// TwinCAT 3 PLC project File
// Title: ZigaLibs.File
// Company: Ziga Javornik
// Author: Ziga Javornik
// ProjectVersion: 0.2.2.0
// Description: Library containing logic for file handling and helper programs.
// ProgramVersion: 3.1.4026.26
// libraries:
//   Tc2_Standard, * (Beckhoff Automation GmbH)
//   Tc2_System, * (Beckhoff Automation GmbH)
//   Tc2_Utilities, * (Beckhoff Automation GmbH)
//   Tc3_Module, * (Beckhoff Automation GmbH)
//   TcError, * (Roald87)
//   TcUnit, * (www.tcunit.org)
//   ZigaLibs.Core, * (Ziga Javornik)
// project tree:
//   SOURCE/Constants/ Constants.TcPOU, FB_PathSeperators.TcPOU, FB_Wildcards.TcPOU
//   SOURCE/DUTs/ E_FileOpenMode.TcDUT, ST_FileInfo.TcDUT, T_FileAccessMode.TcDUT, T_FileHandle.TcDUT
//   SOURCE/Utilities/Directory/ E_DeleteFilesByDateState.TcDUT, E_GetFilesState.TcDUT, FB_DirectoryUtilities.TcPOU, I_Directory.TcIO
//   SOURCE/Utilities/File/ FB_FileUtilities.TcPOU, I_File.TcIO
//   SOURCE/Utilities/Path/ FB_PathGenerator.TcPOU, FB_PathUtilities.TcPOU, I_Path.TcIO, I_PathGenerator.TcIO, I_Wildcards.TcIO
//   SOURCE/FileHandler/ FB_FileHandler.TcPOU, I_FileHandler.TcIO, I_FileProperties.TcIO
//   SOURCE/Utilities/ Utilities.TcPOU
//   / TestsTask.TcTTO
//   TESTS/ PRG_TESTS.TcPOU
//   TESTS/Test suites/ FB_DirectoryUtilities_Tests.TcPOU, FB_FileHandler_Tests.TcPOU, FB_FileUtilities_Tests.TcPOU, FB_Utilities_Tests.TcPOU, FB_PathGenerator_Tests.TcPOU, FB_PathUtilities_Tests.TcPOU
// (motion and I/O tree: see PLC project logging)
// real-time tasks:
//   TASK TestsTask: cycle T#10ms, priority 20, ADS port 350
//   TASK PlcTask: cycle T#10ms, priority 21, ADS port 351

CONFIGURATION File
    RESOURCE PLC ON TwinCAT3
        TASK TestsTask(INTERVAL := T#10ms, PRIORITY := 20);
        PROGRAM PRG_TESTS WITH TestsTask : PRG_TESTS;
    END_RESOURCE
END_CONFIGURATION

// ---- SOURCE/DUTs/E_FileOpenMode.TcDUT
// A combination of file open modes, based on available options.
// Source: https://infosys.beckhoff.com/english.php?content=../content/1033/tcplclib_tc2_system/30977547.html&id=
{attribute 'strict'}
{attribute 'to_string'}
TYPE E_FileOpenMode :
(
	(* r: Opens a file for reading. An error is returned if the file cannot be found or does not exist.*)
	TEXT_READ_MUST_EXIST := Tc2_System.FOPEN_MODEREAD OR Tc2_System.FOPEN_MODETEXT,
	
	(* 	w: Opens an empty file for writing. If the file already exists, it is overwritten.*)
	TEXT_WRITE_OVERWRITE_EXISTING := Tc2_System.FOPEN_MODEWRITE OR Tc2_System.FOPEN_MODETEXT,
	
	(* a: Opens a file for writing at the end of the file (append). If the file does not exist, a new file is created.*)
	TEXT_APPEND := Tc2_System.FOPEN_MODEAPPEND OR Tc2_System.FOPEN_MODETEXT,
	
	(* r+: Opens a file for reading and writing. The file must exist.*)
	TEXT_READ_WRITE_MUST_EXIST := Tc2_System.FOPEN_MODEREAD OR Tc2_System.FOPEN_MODEPLUS OR Tc2_System.FOPEN_MODETEXT,
	
	(* w+: Opens an empty file for reading and writing. If the file already exists, it is overwritten.*)
	TEXT_READ_WRITE_OVERWRITE_EXISTING := Tc2_System.FOPEN_MODEWRITE OR Tc2_System.FOPEN_MODEPLUS OR Tc2_System.FOPEN_MODETEXT,
	
	(* a+: opens a file for reading and writing at the end of the file (append). 
	If the file does not exist, a new file is created. For this, the memory path must be known, otherwise error 1804 appears. 
	All write operations are always performed at end of a file, if the file was opened in the modes a or a+.
	The file pointer can be moved with FB_FileSeek, although for writing it is moved to the end of the file by default, i.e. existing data cannot be overwritten.*)
	TEXT_READ_WRITE_APPEND	:= Tc2_System.FOPEN_MODEAPPEND OR Tc2_System.FOPEN_MODEPLUS OR Tc2_System.FOPEN_MODETEXT,
	
	(* r: Opens a file for reading. An error is returned if the file cannot be found or does not exist.*)
	BINARY_READ_MUST_EXIST	:= Tc2_System.FOPEN_MODEREAD OR Tc2_System.FOPEN_MODEBINARY,
	
	(* 	w: Opens an empty file for writing. If the file already exists, it is overwritten.*)
	BINARY_WRITE_OVERWRITE_EXISTING := Tc2_System.FOPEN_MODEWRITE OR Tc2_System.FOPEN_MODEBINARY,
	
	(* a: Opens a file for writing at the end of the file (append). If the file does not exist, a new file is created.*)
	BINARY_APPEND := Tc2_System.FOPEN_MODEAPPEND OR Tc2_System.FOPEN_MODEBINARY,
	
	(* r+: Opens a file for reading and writing. The file must exist.*)
	BINARY_READ_WRITE_MUST_EXIST := Tc2_System.FOPEN_MODEREAD OR Tc2_System.FOPEN_MODEPLUS OR Tc2_System.FOPEN_MODEBINARY,
	
	(* w+: Opens an empty file for reading and writing. If the file already exists, it is overwritten.*)
	BINARY_READ_WRITE_OVERWRITE_EXISTING := Tc2_System.FOPEN_MODEWRITE OR Tc2_System.FOPEN_MODEPLUS OR Tc2_System.FOPEN_MODEBINARY,
	
	(* a+: opens a file for reading and writing at the end of the file (append). 
	If the file does not exist, a new file is created. For this, the memory path must be known, otherwise error 1804 appears. 
	All write operations are always performed at end of a file, if the file was opened in the modes a or a+.
	The file pointer can be moved with FB_FileSeek, although for writing it is moved to the end of the file by default, i.e. existing data cannot be overwritten.*)
	BINARY_READ_WRITE_APPEND := Tc2_System.FOPEN_MODEAPPEND OR Tc2_System.FOPEN_MODEPLUS OR Tc2_System.FOPEN_MODEBINARY
)DWORD;
END_TYPE

// ---- SOURCE/DUTs/ST_FileInfo.TcDUT
// Structure with all the information for working with file handling..
TYPE ST_FileInfo :
STRUCT
	Handle 		: T_FileHandle;				// File handle
	NetId		: Tc2_System.T_AmsNetID;	// NetId where the file is located
	Name		: Tc2_System.T_MaxString;	// Name of the file
	Path		: Tc2_System.T_MaxString;	// Locaiton of the file
	IsOpened	: BOOL;
END_STRUCT
END_TYPE

// ---- SOURCE/DUTs/T_FileAccessMode.TcDUT
TYPE T_FileAccessMode : DWORD; END_TYPE

// ---- SOURCE/DUTs/T_FileHandle.TcDUT
TYPE T_FileHandle : UINT; END_TYPE

// ---- SOURCE/Utilities/Directory/E_DeleteFilesByDateState.TcDUT
{attribute 'qualified_only'}
{attribute 'strict'}
TYPE E_DeleteFilesByDateState :
(
	START,
	GET_FILE,
	WAIT_FOR_DELETE
);
END_TYPE

// ---- SOURCE/Utilities/Directory/E_GetFilesState.TcDUT
{attribute 'qualified_only'}
{attribute 'strict'}
TYPE INTERNAL E_GetFilesState :
(
	READY,
	START,
	AWAIT_RESULT,
	ALL_FILES_FOUND,
	ERROR
);
END_TYPE

// ---- SOURCE/Utilities/Directory/I_Directory.TcIO
INTERFACE I_Directory

// Deletes files in the directory that were created before the provided date.
METHOD DeleteFilesCreatedBefore : BOOL
VAR_INPUT
	path				: Tc2_System.T_MaxString;	// Path to where the deletion should be performed
	fileNameContains	: Tc2_System.T_MaxString;	// Some characters that the file name should containt
	netId				: Tc2_System.T_AmsNetID;	// NetId where the search should occurr
	thresholdDate		: DT;	// If created before this date, the file will be deleted.
END_VAR

VAR_OUTPUT
	error			: BOOL;
	errorInfo		: ZigaLibs_Core.ST_AdsError;	
	deletedFiles	: ARRAY[0..100] OF Tc2_System.T_MaxString;	// A list of deleted items, as T_MaxString (file names).
END_VAR
END_METHOD

// Looks if the provided directory exists on the disk.
// Returns TRUE when done
// Result can be found in the output directoryExists.
METHOD Exists : BOOL
VAR_INPUT
	directory	: Tc2_System.T_MaxString;	// Path to the directory that will be searched.
	netId		: Tc2_System.T_AmsNetID;	// NetId where to search.
END_VAR

VAR_OUTPUT
	directoryExists		: BOOL;	// TRUE if it exists, else FALSE. Only valid after method returns TRUE.
END_VAR
END_METHOD

(* Looks in the directory `path` and iterates the content. 
 When method returns TRUE, the collection of items is found in the result I_Collection.*)
METHOD ListAll : BOOL
VAR_INPUT
	path	: Tc2_System.T_MaxString;	// Path to the directory that will be searched.
	netId	: Tc2_System.T_AmsNetID;	// NetId where to search.
END_VAR

VAR_IN_OUT
	items	: ARRAY[*] OF Tc2_Utilities.ST_FindFileEntry;	// Collection of found files in the provided location	
END_VAR

VAR_OUTPUT
	error		: BOOL;	// Will be true if an error occurs while executing the file query
	errorInfo	: ZigaLibs_Core.ST_AdsError;	// Error information will be provided here
END_VAR
END_METHOD

(* Looks in the directory `path` and iterates the content. 
 When method returns TRUE, the collection of files is found in the result I_Collection.*)
METHOD ListFiles : BOOL
VAR_INPUT
	path	: Tc2_System.T_MaxString;	// Path to the directory that will be searched.
	netId	: Tc2_System.T_AmsNetID;	// NetId where to search.
END_VAR

VAR_IN_OUT
	files	: ARRAY[*] OF Tc2_System.T_MaxString;	// Collection of found files in the provided location.
END_VAR

VAR_OUTPUT
	error		: BOOL;	// Will be true if an error occurs while executing the file query
	errorInfo	: ZigaLibs_Core.ST_AdsError;	// Error information will be provided here
END_VAR
END_METHOD

END_INTERFACE

// ---- SOURCE/Utilities/File/I_File.TcIO
INTERFACE I_File

METHOD Create : BOOL
VAR_INPUT
	path		: Tc2_System.T_MaxString;	// Path to where the file will be created
	name		: Tc2_System.T_MaxString;	// Name of the file to create.
	netId		: Tc2_System.T_AmsNetID;	// NetId of the device where the file will be created
	overwrite	: BOOL;						// If set to TRUE, if the file with the provided name already exists, it will be overwritten
END_VAR
VAR_OUTPUT
	error			: BOOL;
	errorInfo	: ZigaLibs_Core.ST_AdsError;
END_VAR
END_METHOD

// Deletes the file. Returns TRUE when done.
METHOD Delete : BOOL
VAR_INPUT
	path	: Tc2_System.T_MaxString;	// Location of the file
	name	: Tc2_System.T_MaxString;	// File to be deleted
	netId	: Tc2_System.T_AmsNetID;
END_VAR
VAR_OUTPUT
	error			: BOOL;
	errorInfo	: ZigaLibs_Core.ST_AdsError;
END_VAR
END_METHOD

// Checks the content at `path` and looks for the file with `name`. Returns TRUE when done. 
// If file exissts, the result ˛`result` will be TRUE, else it will be fALSE.
METHOD Exists : BOOL
VAR_INPUT
	path	: Tc2_System.T_MaxString;	// Path to the file location
	name	: Tc2_System.T_MaxString;	// Name of the file
	netId	: Tc2_System.T_AmsNetID;	// NetId where the file is located
END_VAR

VAR_OUTPUT
	result		: BOOL; // Result, if the file exists or not - check when method returns TRUE
	error		: BOOL;	// Will be true if an error occurs while executing the file query
	errorInfo	: ZigaLibs_Core.ST_AdsError; // Error information will be provided here
END_VAR
END_METHOD

END_INTERFACE

// ---- SOURCE/Utilities/Path/I_Path.TcIO
INTERFACE I_Path

(* Checks if path exists, return TRUE when done and the result is returned in `result` output var.*)
METHOD Exists : BOOL
VAR_INPUT
	path	: Tc2_System.T_MaxString;
	netId	: Tc2_System.T_AmsNetID;
END_VAR

VAR_OUTPUT
	result		: BOOL; // Result, if the file exists or not - check when method returns TRUE
	error		: BOOL;	// Will be true if an error occurs while executing the file query
	errorInfo	: ZigaLibs_Core.ST_AdsError; // Error information will be provided here
END_VAR
END_METHOD

(* Generates the file path based on the location, file name and extension*)
METHOD Generate : I_PathGenerator
END_METHOD

END_INTERFACE

// ---- SOURCE/Utilities/Path/I_PathGenerator.TcIO
INTERFACE I_PathGenerator

METHOD AddWildcard : I_Wildcards
VAR_INPUT
END_VAR
END_METHOD

METHOD Create : T_MaxString
VAR_INPUT
END_VAR
END_METHOD

// Concatines the path with previously added paths. 
// If the provided path does not starts with the system-based path seperator, it is added

// Example:
// Join('C:/Program Files/').Join('Utilities/SystemUtilities') 
// will result in 'C:/Program Files/Utilities/SystemUtilities'
METHOD Join : I_PathGenerator
VAR_INPUT
	path	: STRING;
END_VAR
END_METHOD

END_INTERFACE

// ---- SOURCE/Utilities/Path/I_Wildcards.TcIO
INTERFACE I_Wildcards

METHOD Asterisk : I_PathGenerator
VAR_INPUT
	left	: Tc2_System.T_MaxString;
	right	: Tc2_System.T_MaxString;
END_VAR
END_METHOD

METHOD Questionmark : I_PathGenerator
VAR_INPUT
END_VAR
END_METHOD

END_INTERFACE

// ---- SOURCE/FileHandler/I_FileHandler.TcIO
INTERFACE I_FileHandler EXTENDS I_FileProperties

// Closes the file and returns TRUE when done.
METHOD Close : BOOL
END_METHOD

// Creates the file
METHOD Create : BOOL
VAR_INPUT
	path	: Tc2_System.T_MaxString;	// Path to the file location
	name	: Tc2_System.T_MaxString;	// Name of the file
	netId	: Tc2_System.T_AmsNetID;	// NetId where the file is located
END_VAR
END_METHOD

// Flushes the current file stream data to the file. 
// Basically file is closed and re-opened, which in turn writes the content of the stream to the file.
// If the file was opened to overwrite existing content, flushing will clear the data in the file!
// While flushing is being executed, the .File property DOES NOT CHANGE 
// For example, the File.IsOpened will remain TRUE even at the point where it is actually not. It will then be re-opened. 
// If an error occurs however, properties will be set to correct state.

METHOD Flush : BOOL
END_METHOD

// Opens the file in the path provided. If a file is already opened nothing happens.
// Returns: TRUE when done.
METHOD Open : BOOL
VAR_INPUT
	path	: Tc2_System.T_MaxString;	// Path to the file location
	name	: Tc2_System.T_MaxString;	// Name of the file
	mode	: E_FileOpenMode;			// Mode in which the file will be opened
	netId	: Tc2_System.T_AmsNetID;	// NetId where the file is located
END_VAR
END_METHOD

// Opens the last file with the provided open parameters. 
// If file can't be opened or no file has been opened so far, an error is gnerated.
METHOD OpenLast : BOOL
END_METHOD

// Reads the file and writes the content to the result variable.
// Resturns TRUE when done.
METHOD Read : BOOL
VAR_INPUT
	result	: ANY;
END_VAR
END_METHOD

// Reset any existing error.
METHOD Reset
END_METHOD

(* Returns TRUE if there is no content in the file stream.*)
{attribute'monitoring':='call'}
PROPERTY StreamEmpty : BOOL
GET
END_GET
END_PROPERTY

// Writes binary content to the file.
// Returns TRUE when done.
METHOD WriteBinary : BOOL
VAR_INPUT
	data		: ANY;	// Bincary content to be written
END_VAR
END_METHOD

// Writes a single line to the file
// Returns TRUE when done.
METHOD WriteLine : BOOL
VAR_INPUT
	line	: Tc2_System.T_MaxString;	// Text to be written
END_VAR
END_METHOD

END_INTERFACE

// ---- SOURCE/FileHandler/I_FileProperties.TcIO
// Provies interface to properties required for file access
INTERFACE I_FileProperties

{attribute 'monitoring':='call'}
// Gets or set file properties.
PROPERTY File : REFERENCE TO ST_FileInfo
GET
END_GET
END_PROPERTY

END_INTERFACE

// ---- TESTS/PRG_TESTS.TcPOU
PROGRAM INTERNAL PRG_TESTS

(* Instantiate test suites here. Naming convention for tests should be a suffix with _Tests.
Good practice for creating test methods is to end them with _test as well. *)
VAR
	PathGeneratorTests		: FB_PathGenerator_Tests;
	UtilitiesTests			: FB_Utilities_Tests;
	FileHandlerTests		: FB_FileHandler_Tests;
	PathUtilitiesTests		: FB_PathUtilities_Tests;
	FileUtilitiesTests		: FB_FileUtilities_Tests;
	DirectoryUtilitiesTests	: FB_DirectoryUtilities_Tests;
END_VAR

VAR CONSTANT
	FILE_HANDLER_TESTS_PATH			: Tc2_System.T_MaxString := '/home/Administrator/ZigaLibsTestFolder/FileHandlerTests/';
	FILE_HANDLER_TESTS_DIRECTORY	: Tc2_System.T_MaxString := '/home/Administrator/ZigaLibsTestFolder/FileHandlerTests';
	NET_ID							: Tc2_System.T_AmsNetID := '';
	DATE_TIME_MAX_VALUE				: DT  := DATE_AND_TIME#2106-02-07-06:28:15;
END_VAR

// Run tests in parallel
//TcUnit.RUN();

// Run tests in sequence, one after the other.
TcUnit.RUN_IN_SEQUENCE();

END_PROGRAM

// ---- TESTS/Test suites/FB_PathGenerator_Tests.TcPOU
FUNCTION_BLOCK INTERNAL FB_PathGenerator_Tests EXTENDS FB_TestSuite
VAR_INPUT
END_VAR
VAR_OUTPUT
END_VAR
VAR
	_pathGenerator	: FB_PathGenerator;
END_VAR

Test01_VariousPathOptions();

METHOD Test01_VariousPathOptions

// These test values were taken from microsoft Path.Join documentation at 
// https://learn.microsoft.com/en-us/dotnet/api/system.io.path.join?view=net-9.0
VAR
	path1 : STRING := 'C:/Program Files/';
	path2 : STRING := 'Utilities/SystemUtilities';
	expectedResult_path1_2	: STRING := 'C:/Program Files/Utilities/SystemUtilities';
	
	
	path3 : STRING := 'C:/';
	path4 : STRING := '/Program Files';
	expectedResult_path3_4	: STRING := 'C://Program Files';
	
	path5 : STRING := 'C:/Users/Public/Documents/';
	path6 : STRING := 'C:/Users/User1/Documents/Financial/';
	expectedResult_path5_6	: STRING := 'C:/Users/Public/Documents/C:/Users/User1/Documents/Financial/';	
END_VAR
TcUnit.TEST('Test01_VariousPathOptions');

AssertEquals_STRING(
	Expected := expectedResult_path1_2, 
	Actual := _pathGenerator.Join(path1).Join(path2).Create(),
	'Joining paths 1 and 2 failed.');
	
AssertEquals_STRING(
	Expected := expectedResult_path3_4, 
	Actual := _pathGenerator.Join(path3).Join(path4).Create(),
	'Joining paths 2 and 3 failed.');
	
AssertEquals_STRING(
	Expected := expectedResult_path5_6, 
	Actual := _pathGenerator.Join(path5).Join(path6).Create(),
	'Joining paths 4 and 5 failed.');
		
TcUnit.TEST_FINISHED();
END_METHOD

END_FUNCTION_BLOCK

// ---- SOURCE/Utilities/Path/FB_PathGenerator.TcPOU
FUNCTION_BLOCK FB_PathGenerator IMPLEMENTS I_PathGenerator, I_Wildcards
VAR_INPUT
END_VAR
VAR_OUTPUT
END_VAR
VAR
	_path			: Tc2_System.T_MaxString;
END_VAR

// Provides ability to add allowed wildcards to the generating path.
METHOD AddWildcard : I_Wildcards
AddWildcard := THIS^;
END_METHOD

// Adds the asterisk (*) wildcard between the left and right strings provided
// Example Asterix('abc','def') => '<path so far>abc*def'
METHOD Asterisk : I_PathGenerator
VAR_INPUT
	left	: Tc2_System.T_MaxString;
	right	: Tc2_System.T_MaxString;
END_VAR
ZigaLibs_Core.StringHelper.Join(left, Constants.Wildcards.Asterisk);
ZigaLibs_Core.StringHelper.Join(left, right);
ZigaLibs_Core.StringHelper.Join(_path, left);
Asterisk := THIS^;
END_METHOD

METHOD Create : Tc2_System.T_MaxString
Create := _path;
_path := '';
END_METHOD

// Concatines the path with previously added paths. 
// If the provided path does not starts with the system-based path seperator, it is added

// Example:
// Join('C:/Program Files/').Join('Utilities/SystemUtilities') 
// will result in 'C:/Program Files/Utilities/SystemUtilities'
METHOD Join : I_PathGenerator
VAR_INPUT
	path	: STRING;
END_VAR
Join := THIS^;

// If this is the root, skip adding seperator to start.
IF Tc2_Standard.FIND(path, ':') <> 0 THEN
	ZigaLibs_Core.StringHelper.Join(_path, path);
	RETURN;
END_IF

// Add path seperator, if not starting with it.
IF NOT ZigaLibs_Core.StringHelper.StartsWith(path, Constants.PathSeperators.Windows) AND
   NOT ZigaLibs_Core.StringHelper.EndsWith(_path, Constants.PathSeperators.Windows) AND
   NOT ZigaLibs_Core.StringHelper.StartsWith(path, Constants.PathSeperators.Unix) AND
   NOT ZigaLibs_Core.StringHelper.EndsWith(_path, Constants.PathSeperators.Unix)
THEN
	path := Tc2_Standard.CONCAT(Constants.PathSeperators.Independent, path);
END_IF
ZigaLibs_Core.StringHelper.Join(_path, path);
END_METHOD

// Adds the question mark (?) wildcard to the end of the currently generated path.
METHOD Questionmark : I_PathGenerator
ZigaLibs_Core.StringHelper.Join(_path, Constants.Wildcards.QuestionMark);
Questionmark := THIS^;
END_METHOD

END_FUNCTION_BLOCK

// ---- SOURCE/Constants/Constants.TcPOU
// Contains string constants for working with files
{attribute 'no_explicit_call' := 'Body contains no logic, calling methods only allowed.'}
{attribute 'hide_all_locals'}
PROGRAM Constants
VAR
	_pathSeperators	: FB_PathSeperators;	
	_wildcards	: FB_Wildcards;
END_VAR

// Returns WINDOWS path separator "/"
PROPERTY PathSeperators : REFERENCE TO FB_PathSeperators
GET
PathSeperators REF= _pathSeperators;
END_GET
END_PROPERTY

PROPERTY Wildcards : REFERENCE TO FB_Wildcards
GET
Wildcards REF= _wildcards;
END_GET
END_PROPERTY

END_PROGRAM

// ---- SOURCE/Constants/FB_PathSeperators.TcPOU
{attribute 'no_explicit_call' := 'Body contains no logic, calling methods only allowed.'}
FUNCTION_BLOCK INTERNAL FB_PathSeperators
VAR_INPUT
END_VAR
VAR_OUTPUT
END_VAR
VAR
END_VAR

PROPERTY Independent : T_Char
GET
Independent := '/';
END_GET
END_PROPERTY

PROPERTY PUBLIC Unix : T_Char
GET
Unix := '\';
END_GET
END_PROPERTY

PROPERTY Windows : T_Char
GET
Windows := '/';
END_GET
END_PROPERTY

END_FUNCTION_BLOCK

// ---- SOURCE/Constants/FB_Wildcards.TcPOU
{attribute 'no_explicit_call' := 'Body contains no logic, calling methods only allowed.'}
FUNCTION_BLOCK INTERNAL FB_Wildcards

// Matches any number of characters. You can use the asterisk (*) anywhere in a character string.
// Example: wh* finds what, white, and why, but not awhile or watch.
PROPERTY Asterisk : ZigaLibs_Core.T_Char
GET
Asterisk := '*';
END_GET
END_PROPERTY

// Matches a single alphabet in a specific position.
// Example: b?ll finds ball, bell, and bill.
PROPERTY QuestionMark : ZigaLibs_Core.T_Char
GET
QuestionMark := '?';
END_GET
END_PROPERTY

END_FUNCTION_BLOCK

// ---- SOURCE/Utilities/Utilities.TcPOU
// A class with helper methods when working with files.
{attribute 'no_explicit_call' := 'Body contains no logic, calling methods only allowed.'}
PROGRAM Utilities

VAR
	_directory	: FB_DirectoryUtilities;
	_file		: FB_FileUtilities;
	_path		: FB_PathUtilities;
END_VAR

PROPERTY Directory : I_Directory
GET
Directory := _directory;
END_GET
END_PROPERTY

PROPERTY File : I_File
GET
File := _file;
END_GET
END_PROPERTY

PROPERTY Path : I_Path
GET
Path := _path;
END_GET
END_PROPERTY

END_PROGRAM

// ---- SOURCE/Utilities/Directory/FB_DirectoryUtilities.TcPOU
FUNCTION_BLOCK FB_DirectoryUtilities IMPLEMENTS I_Directory
VAR_INPUT
END_VAR
VAR_OUTPUT
END_VAR
VAR
END_VAR

// Deletes matching files in the directory that were created before the provided date.
METHOD DeleteFilesCreatedBefore : BOOL
VAR_INPUT
	path				: Tc2_System.T_MaxString;	// Path to where the deletion should be performed
	fileNameContains	: Tc2_System.T_MaxString;	// Some characters that the file name should containt
	netId				: Tc2_System.T_AmsNetID;	// NetId where the search should occurr
	thresholdDate		: DT;	// If created before this date, the file will be deleted.
END_VAR
VAR_OUTPUT
	error			: BOOL;
	errorInfo		: ZigaLibs_Core.ST_AdsError;	
	deletedFiles	: ARRAY[0..100] OF Tc2_System.T_MaxString;	// A list of deleted items, as T_MaxString (file names).
END_VAR

VAR_INST
	files				: ARRAY[0..100] OF Tc2_Utilities.ST_FindFileEntry;
	currentFile			: ST_FindFileEntry;
	state				: E_DeleteFilesByDateState;
	fileUtilities		: FB_FileUtilities;
	deleteFilesLocal	: ARRAY[0..100] OF Tc2_System.T_MaxString;
	fileIndex			: DINT;
END_VAR
VAR
	timeOfCreation		: DT;
	deletedFileIndex	: ZigaLibs_Core.T_ArrayIndexer;
END_VAR
CASE state OF
	E_DeleteFilesByDateState.START:
		fileIndex := 0;
		IF THIS^.ListAll(path := path, netId := netId, items := files, error => error, errorInfo => errorInfo) THEN
			state := E_DeleteFilesByDateState.GET_FILE;
		END_IF
	
	E_DeleteFilesByDateState.GET_FILE:
		// Iterate the array, delete files that match the criteria - name contains the string and it was created before date
		
		IF fileIndex <= 100 AND fileIndex >= 0 THEN
			currentFile := files[fileIndex];
			fileIndex := fileIndex + 1;
			IF currentFile.sFileName <> '' AND_THEN Tc2_Standard.FIND(currentFile.sFileName, fileNameContains) <> 0 THEN
				// Matching file found, check date of creation
				timeOfCreation := Tc2_Utilities.FILETIME_TO_DT(currentFile.creationTime);
				IF timeOfCreation < thresholdDate THEN
					// Date is lower than provided date threshold
					state := E_DeleteFilesByDateState.WAIT_FOR_DELETE;
				END_IF
			END_IF 
		ELSE
			deletedFiles := deleteFilesLocal;
			state := E_DeleteFilesByDateState.START;
			DeleteFilesCreatedBefore := TRUE;
		END_IF
	
	E_DeleteFilesByDateState.WAIT_FOR_DELETE:
		IF fileUtilities.Delete(
			path, 
			currentFile.sFileName, 
			netId, 
			error => error, errorInfo => errorInfo) 
		THEN
			IF error THEN
				DeleteFilesCreatedBefore := TRUE;
				RETURN;
			END_IF
			ZigaLibs_Core.ArrayHelper.ShiftUp(deletedFiles, deleteFilesLocal[0]);
			deleteFilesLocal[0] := currentFile.sFileName;
			state := E_DeleteFilesByDateState.GET_FILE;
		END_IF
END_CASE
END_METHOD

(* Looks if the provided directory exists on the disk.
 Returns TRUE when done
 Result can be found in the output directoryExists.*)
METHOD Exists : BOOL
VAR_INPUT
	(* Path to the directory that will be searched.*)
	directory	: Tc2_System.T_MaxString;
	(* NetId where to search.*)
	netId	: Tc2_System.T_AmsNetID;
END_VAR
VAR_OUTPUT
	(* TRUE if it exists, else FALSE. Only valid after method returns TRUE.*)
	directoryExists	: BOOL;
END_VAR

VAR
	foundItems 			: ARRAY[0..100] OF Tc2_Utilities.ST_FindFileEntry;
	currentItemIndex	: ZigaLibs_Core.T_ArrayIndexer;
	currentItem			: Tc2_Utilities.ST_FindFileEntry;
	directoryName		: Tc2_System.T_MaxString;
	charPosiiton		: INT;
	itemName			: Tc2_System.T_MaxString;
END_VAR
// List all the items...
IF THIS^.ListAll(path := directory, netId := netId, items := foundItems) THEN
	// Split the path into directories
	
	WHILE Tc2_Standard.FIND(STR1 := directoryName, STR2 := '.') <> 0 DO
		charPosiiton := Tc2_Standard.FIND(directoryName, '.');
		directoryName := Tc2_Standard.DELETE(directoryName, charPosiiton, 1);
	END_WHILE

	// Iterate the returned items and check if it is directory and the name is correct. Exit on success.
	FOR currentItemIndex := 0 TO 100 BY 1 DO
		currentItem := foundItems[currentItemIndex];
		IF currentItem.fileAttributes.bDirectory AND_THEN
			currentItem.sFileName = directoryName
		THEN
			directoryExists := TRUE;
			EXIT;
		END_IF
	END_FOR
END_IF

Exists := TRUE;
END_METHOD

(* Looks in the directory `path` and iterates the content. 
 When method returns TRUE, the collection of items is found in the result I_Collection.*)
METHOD ListAll : BOOL
VAR_INPUT
	path	: Tc2_System.T_MaxString;	// Path to the directory that will be searched.
	netId	: Tc2_System.T_AmsNetID;	// NetId where to search.
END_VAR

VAR_IN_OUT
	items	: ARRAY[*] OF Tc2_Utilities.ST_FindFileEntry;	// Collection of found files in the provided location	
END_VAR

VAR_OUTPUT
	error		: BOOL;	// Will be true if an error occurs while executing the file query
	errorInfo	: ZigaLibs_Core.ST_AdsError;	// Error information will be provided here
END_VAR

VAR_INST
	fbFindFileEntries	: Tc2_Utilities.FB_EnumFindFileEntry;
	eGetFilesState		: E_GetFilesState;
	itemsArrayIndex		: ZigaLibs_Core.T_ArrayIndexer;
END_VAR

VAR
	varInfo	: ZigaLibs_Core.T_VarInfo;
END_VAR
CASE eGetFilesState OF
	
	E_GetFilesState.READY:
		fbFindFileEntries(bExecute := FALSE, 
		eCmd := Tc2_Utilities.E_EnumCmdType.eEnumCmd_First);
		// Clear the array when startin
		Tc2_System.MEMSET(destAddr := ADR(items[0]), fillByte := 0, n := SIZEOF(items));
		itemsArrayIndex := 0;	
		eGetFilesState := E_GetFilesState.START;

	E_GetFilesState.START:
		error := FALSE;
		errorInfo.Code := 0;
		errorInfo.Source := '';
		
		// Path/* returns all entries
		fbFindFileEntries(bExecute := TRUE, sNetId := netId,
			sPathName := Utilities.Path.Generate()
				.Join(path)
				.AddWildcard().Asterisk(left := '', right :='')
				.Create());
			
		eGetFilesState := E_GetFilesState.AWAIT_RESULT;
	
	E_GetFilesState.AWAIT_RESULT:
		fbFindFileEntries(bExecute := FALSE);
		
		IF fbFindFileEntries.bError THEN
			eGetFilesState := E_GetFilesState.ERROR;
			RETURN;
		END_IF
		
		IF fbFindFileEntries.bBusy THEN
			RETURN;
		END_IF
		
		IF NOT fbFindFileEntries.bEOE AND (itemsArrayIndex <= UPPER_BOUND(items, 1)) THEN
			items[itemsArrayIndex] := fbFindFileEntries.stFindFile;
			itemsArrayIndex := itemsArrayIndex + 1;
			fbFindFileEntries.eCmd := Tc2_Utilities.E_EnumCmdType.eEnumCmd_Next;
			eGetFilesState := E_GetFilesState.START;
			RETURN;
		END_IF
		
		eGetFilesState := E_GetFilesState.ALL_FILES_FOUND;
	
	E_GetFilesState.ALL_FILES_FOUND:
		ListAll := TRUE;
		eGetFilesState := E_GetFilesState.READY;
		
	E_GetFilesState.ERROR:
		error := TRUE;
		errorInfo.Code := TcError.ToAdsErrorCode(fbFindFileEntries.nErrID);
		varInfo := __VARINFO(fbFindFileEntries);
		errorInfo.Source := varInfo.Symbol;
		
		ListAll := TRUE;
		eGetFilesState := E_GetFilesState.READY;
END_CASE
END_METHOD

(* Looks in the directory `path` and iterates the content. 
 When method returns TRUE, the collection of files is found in the result I_Collection.*)
METHOD ListFiles : BOOL
VAR_INPUT
	path	: Tc2_System.T_MaxString;	// Path to the directory that will be searched.
	netId	: Tc2_System.T_AmsNetID;	// NetId where to search.
END_VAR

VAR_IN_OUT
	files	: ARRAY[*] OF Tc2_System.T_MaxString;	// Collection of found files in the provided location.
END_VAR

VAR_OUTPUT
	error		: BOOL;	// Will be true if an error occurs while executing the file query
	errorInfo	: ZigaLibs_Core.ST_AdsError;	// Error information will be provided here
END_VAR

VAR_INST
	fbFindFileEntries	: Tc2_Utilities.FB_EnumFindFileEntry;
	eGetFilesState		: E_GetFilesState;
	filesArrayIndex		: ZigaLibs_Core.T_ArrayIndexer;
END_VAR

VAR
	varInfo	: ZigaLibs_Core.T_VarInfo;
END_VAR
CASE eGetFilesState OF
	
	E_GetFilesState.READY:
		fbFindFileEntries(bExecute := FALSE, 
			eCmd := Tc2_Utilities.E_EnumCmdType.eEnumCmd_First);
		Tc2_System.MEMSET(destAddr := files, fillByte := 0, n := SIZEOF(files));		
		filesArrayIndex := 0;
		eGetFilesState := E_GetFilesState.START;

	E_GetFilesState.START:
		error := FALSE;
		errorInfo.Code := 0;
		errorInfo.Source := '';
		
		// Path/*.* returns all files
		fbFindFileEntries(bExecute := TRUE, sNetId := netId,
			sPathName := Utilities.Path.Generate()
				.Join(path)
				.AddWildcard().Asterisk('','')
				.AddWildcard().Asterisk('.', '')
				.Create());
			
		eGetFilesState := E_GetFilesState.AWAIT_RESULT;
	
	E_GetFilesState.AWAIT_RESULT:
		fbFindFileEntries(bExecute := FALSE);
		
		IF fbFindFileEntries.bError THEN
			eGetFilesState := E_GetFilesState.ERROR;
			RETURN;
		END_IF
		
		IF fbFindFileEntries.bBusy THEN
			RETURN;
		END_IF
		
		IF NOT fbFindFileEntries.bEOE AND (filesArrayIndex <= UPPER_BOUND(files, 1)) THEN
			files[filesArrayIndex] := fbFindFileEntries.stFindFile.sFileName;
			filesArrayIndex := filesArrayIndex + 1;
			fbFindFileEntries.eCmd := Tc2_Utilities.E_EnumCmdType.eEnumCmd_Next;
			eGetFilesState := E_GetFilesState.START;
			RETURN;
		END_IF
		
		eGetFilesState := E_GetFilesState.ALL_FILES_FOUND;
	
	E_GetFilesState.ALL_FILES_FOUND:
		ListFiles := TRUE;
		eGetFilesState := E_GetFilesState.READY;
		
	E_GetFilesState.ERROR:
		error := TRUE;
		errorInfo.Code := TcError.ToAdsErrorCode(fbFindFileEntries.nErrID);
		varInfo := __VARINFO(fbFindFileEntries);
		errorInfo.Source := varInfo.Symbol;
		
		ListFiles := TRUE;
		eGetFilesState := E_GetFilesState.READY;
END_CASE
END_METHOD

END_FUNCTION_BLOCK

// ---- SOURCE/Utilities/File/FB_FileUtilities.TcPOU
// Provides file functionalities.
FUNCTION_BLOCK FB_FileUtilities IMPLEMENTS I_File

METHOD Create : BOOL
VAR_INPUT
	(* Path to where the file will be created*)
	path	: Tc2_System.T_MaxString;
	(* Name of the file to create.*)
	name	: Tc2_System.T_MaxString;
	(* NetId of the device where the file will be created*)
	netId	: Tc2_System.T_AmsNetID;
	(* If set to TRUE, if the file with the provided name already exists, it will be overwritten*)
	overwrite	: BOOL;
END_VAR

VAR_OUTPUT
	error			: BOOL;
	errorInfo	: ZigaLibs_Core.ST_AdsError;
END_VAR

VAR_INST
	fbFileHandler	: FB_FileHandler;
	mode			: E_FileOpenMode;
END_VAR
IF overwrite THEN
	mode := E_FileOpenMode.BINARY_READ_WRITE_APPEND;
ELSE
	mode := E_FileOpenMode.BINARY_APPEND;
END_IF

IF NOT fbFileHandler.File.IsOpened THEN
fbFileHandler.Open(
	mode := mode, 
	name := name, 
	netId := netId, 
	path := path);
ELSE
	Create := fbFileHandler.Close();
END_IF

error := fbFileHandler.Error;
errorInfo := fbFileHandler.AdsError;
END_METHOD

(* Deletes the file. Returns TRUE when done.*)
METHOD Delete : BOOL
VAR_INPUT
	(* Location of the file*)
	path	: Tc2_System.T_MaxString;
	(* File to be deleted*)
	name	: Tc2_System.T_MaxString;
	netId	: Tc2_System.T_AmsNetID;
END_VAR
VAR_OUTPUT
	error		: BOOL;
	errorInfo	: ZigaLibs_Core.ST_AdsError;
END_VAR

VAR_INST
	fbFileDelete	: Tc2_System.FB_FileDelete;
END_VAR
fbFileDelete(
	sPathName := Utilities.Path.Generate().Join(path).Join(name).Create(),
	sNetId := netId,
	bExecute := NOT fbFileDelete.bBusy);
	
error := fbFileDelete.bError;
errorInfo.Code := TcError.ToAdsErrorCode(fbFileDelete.nErrId);
errorInfo.Message := TcError.AdsErrorCodeDescription(errorInfo.Code);
	
IF NOT fbFileDelete.bBusy THEN
	fbFileDelete(bExecute := FALSE);
	Delete := TRUE;
END_IF
END_METHOD

(* Checks the content at `path` and looks for the file with `name`. Returns TRUE when done. 
 If file exissts, the result ˛`result` will be TRUE, else it will be fALSE.*)
METHOD Exists : BOOL
VAR_INPUT
	path	: Tc2_System.T_MaxString;	// Path to the file location
	name	: Tc2_System.T_MaxString;	// Name of the file
	netId	: Tc2_System.T_AmsNetID;	// NetId where the file is located
END_VAR

VAR_OUTPUT
	result		: BOOL; // Result, if the file exists or not - check when method returns TRUE
	error		: BOOL;	// Will be true if an error occurs while executing the file query
	errorInfo	: ZigaLibs_Core.ST_AdsError; // Error information will be provided here
END_VAR
	
VAR_INST
	foundFiles			: ARRAY[0..100] OF Tc2_System.T_MaxString;
END_VAR

VAR
	index	: ZigaLibs_Core.T_ArrayIndexer;
END_VAR
IF Utilities.Directory.ListFiles(path := path, netId := netId, files := foundFiles) THEN
	Exists := TRUE;
	FOR index := 0 TO 100 BY 1 DO
		IF foundFiles[index] = name THEN
			result := TRUE;
			RETURN;
		END_IF
	END_FOR
END_IF
END_METHOD

END_FUNCTION_BLOCK

// ---- SOURCE/FileHandler/FB_FileHandler.TcPOU
// A function block containing multiple file handling methods. 
// Note that the body of this FB does NOT need to be called as it holds no logic.
// All the methods should be called untill they return true, if they provide error information, 
// it will be trough a reference variable.
//
// For examples refer to tests in the folder "TESTS/Test suites", file "FB_FileHandlerTests".

{attribute 'no_explicit_call' := 'Body contains no logic, calling methods only allowed.'}
FUNCTION_BLOCK FB_FileHandler EXTENDS ZigaLibs_Core.FB_ErrorSource IMPLEMENTS I_FileHandler

VAR
	_fileInfo		: ST_FileInfo;
	_netId			: Tc2_System.T_AmsNetID;
	_lastOpenMode	: E_FileOpenMode;
	_streamEmpty	: BOOL := TRUE;
END_VAR

// Closes the file and returns TRUE when done.
METHOD Close : BOOL
Close := THIS^.CloseSilent(FALSE);
END_METHOD

// Closes the file without clearing the file properties.
METHOD PRIVATE CloseSilent : BOOL
VAR_INPUT
	silent	: BOOL; // IF set to TRUE, the file property won't be modified. To be used when flushing the stream.
END_VAR
VAR_INST
	fbFileClose	: Tc2_System.FB_FileClose;
END_VAR

VAR
	varInfo	: ZigaLibs_Core.T_VarInfo;
END_VAR
fbFileClose(
	bExecute := NOT fbFileClose.bBusy,
	hFile := File.Handle,
	sNetId := File.NetId);

IF NOT fbFileClose.bBusy THEN
	CloseSilent := TRUE;
	IF fbFileClose.bError THEN
		varInfo := __VARINFO(fbFileClose);
		THIS^.RaiseAdsError(Tc2_Standard.CONCAT(THIS^.InstancePath, varInfo.Symbol), fbFileClose.nErrId);
		THIS^.GenericError.Message := Tc2_Standard.CONCAT('An error occured when closing the file ', File.Name);
		fbFileClose(bExecute := FALSE);	
		RETURN;
	END_IF
	
	_streamEmpty := TRUE;
	fbFileClose(bExecute := FALSE);
	File.Handle := 0;	
	IF NOT silent THEN
		File.IsOpened := FALSE;
	END_IF
END_IF
END_METHOD

// Creates the file, if it does not yet exist,
METHOD Create : BOOL
VAR_INPUT
	path	: Tc2_System.T_MaxString;	// Path to the file location
	name	: Tc2_System.T_MaxString;	// Name of the file
	netId	: Tc2_System.T_AmsNetID;	// NetId where the file is located
END_VAR
VAR
	sb	: ZigaLibs_Core.FB_StringBuilder;
END_VAR
IF NOT file.IsOpened THEN
	THIS^.Open(
		path := path,
		name := name,
		mode := E_FileOpenMode.BINARY_APPEND,
		netId := netId);
		
	// Error opening the file, report and stop.
	IF THIS^.Error THEN
		THIS^.GenericError.Source := sb.Reset()
			.AddString(THIS^.InstancePath)
			.AddString('.Create()')
			.Create();
		
		THIS^.GenericError.Message := sb.Reset()
			.AddString('An error occurred when creating the file, while opening it:')
			.AddString(' Path = ').AddWithDblQuotationMarks(path)
			.AddString(' Name = ').AddWithDblQuotationMarks(name)
			.AddString(' NetId = ').AddWithDblQuotationMarks(netId)
			.AddString('. Refer to AdsError for more info.')
			.Create();
		Create := TRUE;
		RETURN;
	END_IF
ELSE
	Create := THIS^.Close();
	
	// Error closing the file. Report and stop.
	IF THIS^.Error THEN
		THIS^.GenericError.Source := sb.Reset()
			.AddString(THIS^.InstancePath)
			.AddString('.Create()')
			.Create();
		THIS^.GenericError.Message := sb.Reset()
			.AddString('An error occurred when creating the file, while closing it:')
			.AddString(' Path = ').AddWithDblQuotationMarks(path)
			.AddString(' Name = ').AddWithDblQuotationMarks(name)
			.AddString(' NetId = ').AddWithDblQuotationMarks(netId)
			.AddString('. Refer to AdsError for more info.')
			.Create();
	END_IF
END_IF
END_METHOD

{attribute 'monitoring':='call'}
(* Gets the current file properties.*)
PROPERTY File : REFERENCE TO ST_FileInfo
GET
File REF= _fileInfo;
END_GET
END_PROPERTY

// Flushes the current file stream data to the file. 
// Basically file is closed and re-opened, which in turn writes the content of the stream to the file.
// If the file was opened to overwrite existing content, flushing will clear the data in the file!
// While flushing is being executed, the .File property DOES NOT CHANGE 
// For example, the File.IsOpened will remain TRUE even at the point where it is actually not. It will then be re-opened. 
// If an error occurs however, properties will be set to correct state.

METHOD Flush : BOOL
VAR_INST
	closeDone		: BOOL;
END_VAR
IF closeDone OR_ELSE THIS^.CloseSilent(TRUE) THEN
	// Error closing the file while flushing...
	IF THIS^.Error AND NOT closeDone THEN
		Flush := TRUE;
		THIS^.GenericError.Message := 'An error occurred while flushing the file stream (closing the file)...';
		THIS^.GenericError.Source := Tc2_Standard.CONCAT(THIS^.InstanceName, '.Flush()');
		RETURN;
	END_IF
	
	closeDone := TRUE;
END_IF

IF closeDone AND_THEN THIS^.Open(File.Path, File.Name, _lastOpenMode, File.NetId) THEN
	closeDone := FALSE;
	Flush := TRUE;
	// Error while opening the file while flushing...
	IF THIS^.Error THEN
		THIS^.File.Handle := 0;
		THIS^.File.IsOpened := FALSE;
		THIS^.GenericError.Message := 'An error occurred while flushing the file stream (opening the file)...';
		THIS^.GenericError.Source := Tc2_Standard.CONCAT(THIS^.InstanceName, '.Flush()');
	END_IF
END_IF
END_METHOD

// Opens the file in the path provided. If a file is already opened nothing happens.
// Returns: TRUE when done.
METHOD Open : BOOL
VAR_INPUT
	path	: Tc2_System.T_MaxString;	// Path to the file location
	name	: Tc2_System.T_MaxString;	// Name of the file
	mode	: E_FileOpenMode;			// Mode in which the file will be opened
	netId	: Tc2_System.T_AmsNetID;	// NetId where the file is located
END_VAR

VAR_INST
	fbFileOpen	: Tc2_System.FB_FileOpen;
END_VAR

VAR
	varInfo	: ZigaLibs_Core.T_VarInfo;
END_VAR
IF THIS^.File.Handle <> 0 THEN
	Open := TRUE;
	RETURN;
END_IF

fbFileOpen(
	bExecute := NOT fbFileOpen.bBusy,
	nMode := mode,
	sNetId := netID,
	sPathName := Utilities.Path.Generate().Join(path).Join(name).Create());
	
IF NOT fbFileOpen.bBusy THEN
	Open := TRUE;
	IF fbFileOpen.bError THEN
		varInfo := __VARINFO(fbFileOpen);
		THIS^.RaiseAdsError(Tc2_Standard.CONCAT(THIS^.InstancePath, varInfo.Symbol), fbFileOpen.nErrId);
		fbFileOpen(bExecute := FALSE);
		RETURN;
	END_IF
	_lastOpenMode := mode;
	fbFileOpen(bExecute := FALSE);
	File.Handle := fbFileOpen.hFile;
	File.Name := name;
	File.Path := path;
	File.NetId := netId;
	File.IsOpened := TRUE;
END_IF
END_METHOD

(* Opens the last file with the provided open parameters. 
 If file can't be opened or no file has been opened so far, an error is gnerated.*)
METHOD OpenLast : BOOL
IF File.Name = '' THEN
	THIS^.Error := TRUE;
	THIS^.GenericError.Message := 'Can not open file - name is empty.';
	THIS^.GenericError.Source := Tc2_Standard.CONCAT(THIS^.InstanceName, '.OpenLast()');
	OpenLast := TRUE;
	RETURN;
ELSIF File.Path = '' THEN
	THIS^.Error := TRUE;
	THIS^.GenericError.Message := 'Can not open file - path is empty.';
	THIS^.GenericError.Source := Tc2_Standard.CONCAT(THIS^.InstanceName, '.OpenLast()');	
	OpenLast := TRUE;
	RETURN;
ELSIF _lastOpenMode = 0 THEN
	THIS^.Error := TRUE;
	THIS^.GenericError.Message := Tc2_Standard.CONCAT('Can not open file - incorrect file open mode used: ', TO_STRING(_lastOpenMode));
	THIS^.GenericError.Source := Tc2_Standard.CONCAT(THIS^.InstanceName, '.OpenLast()');	
	OpenLast := TRUE;
	RETURN;
ELSIF File.IsOpened THEN
	THIS^.Error := TRUE;
	THIS^.GenericError.Message := 'Can not open last file - file already opened!';
	THIS^.GenericError.Source := Tc2_Standard.CONCAT(THIS^.InstanceName, '.OpenLast()');	
	OpenLast := TRUE;
	RETURN;	
END_IF

IF THIS^.Open(File.Path, File.Name, _lastOpenMode, File.NetId) THEN
	OpenLast := TRUE;
	IF THIS^.Error THEN
		THIS^.GenericError.Message := 'An error has occurred while attempting to open the last opened file. Refer to AdsError for more info.';
		THIS^.GenericError.Source := Tc2_Standard.CONCAT(THIS^.InstanceName, '.OpenLast()');	
	END_IF
END_IF
END_METHOD

// Raise an error for a certain FB instance (calls from methods)
METHOD PROTECTED RaiseAdsError : BOOL
VAR_INPUT
	source	: STRING;
	code 	: UDINT;
END_VAR
THIS^.AdsError.Code := TcError.ToAdsErrorCode(code);
THIS^.AdsError.Source := source;
THIS^.Error := TRUE;
END_METHOD

// Reads the file and writes the content to the result variable.
// Returns TRUE when done.
METHOD Read : BOOL

VAR_INPUT
	result	: ANY;
END_VAR

VAR_INST
	fbFileRead	: Tc2_System.FB_FileRead;
END_VAR

VAR
	varInfo	: ZigaLibs_Core.T_VarInfo;
END_VAR
fbFileRead(
	bExecute := NOT fbFileRead.bBusy,
	sNetId := THIS^.File.NetId,
	hFile := THIS^.File.Handle,
	pReadBuff := result.pValue,
	cbReadLen := DINT_TO_UDINT(result.diSize));
	
IF NOT fbFileRead.bBusy THEN
	Read := TRUE;
	IF fbFileRead.bError THEN
		varInfo := __VARINFO(fbFileRead);
		THIS^.GenericError.Message := Tc2_Standard.CONCAT('An error occured when reading the file ', File.Name);
		THIS^.RaiseAdsError(Tc2_Standard.CONCAT(THIS^.InstancePath, varInfo.Symbol), fbFileRead.nErrId);
		fbFileRead(bExecute := FALSE);
	END_IF
END_IF
END_METHOD

// Reset any existing error.
METHOD Reset
THIS^.ResetError();
END_METHOD

(* Returns TRUE if there is no content in the file stream.*)
{attribute'monitoring':='call'}
PROPERTY StreamEmpty : BOOL
GET
StreamEmpty := _streamEmpty;
END_GET
END_PROPERTY

// Writes binary content to the file.
// Returns TRUE when done.
METHOD WriteBinary : BOOL

VAR_INPUT
	data		: ANY;	// Bincary content to be written
END_VAR

VAR_INST
	fbFileWrite		: Tc2_System.FB_FileWrite;
END_VAR
VAR
	varInfo	: ZigaLibs_Core.T_VarInfo;
END_VAR
_streamEmpty := FALSE;

fbFileWrite(
	bExecute := NOT fbFileWrite.bBusy,
	sNetId := File.NetId,
	hFile := File.Handle,
	pWriteBuff := data.pValue,
	cbWriteLen := DINT_TO_UDINT(data.diSize));
	
IF NOT fbFileWrite.bBusy THEN
	IF fbFileWrite.bError THEN
		varInfo := __VARINFO(fbFileWrite);
		THIS^.RaiseAdsError(Tc2_Standard.CONCAT(THIS^.InstancePath, varInfo.Symbol), fbFileWrite.nErrId);
		WriteBinary := TRUE;
		fbFileWrite(bExecute := FALSE);
		RETURN;
	END_IF
	WriteBinary := TRUE;
	fbFileWrite(bExecute := FALSE);
	_streamEmpty := FALSE;
END_IF
END_METHOD

// Writes a single line to the file
// Returns TRUE when done.
METHOD WriteLine : BOOL

VAR_INPUT
	line : Tc2_System.T_MaxString;	// Text to be written
END_VAR

VAR_INST
	fbFilePuts 		: Tc2_System.FB_FilePuts;
END_VAR

VAR
	varInfo	: ZigaLibs_Core.T_VarInfo;
END_VAR
fbFilePuts(
	bExecute := NOT fbFilePuts.bBusy,
	sNetId := File.NetId,
	hFile := File.Handle,
	sLine := line);
	
IF NOT fbFilePuts.bBusy THEN
	IF fbFilePuts.bError THEN
		varInfo := __VARINFO(fbFilePuts);
		THIS^.RaiseAdsError(Tc2_Standard.CONCAT(THIS^.InstancePath, varInfo.Symbol), fbFilePuts.nErrId);
		fbFilePuts(bExecute := FALSE);
		WriteLine := TRUE;
		RETURN;
	END_IF
	_streamEmpty := FALSE;
	WriteLine := TRUE;
	fbFilePuts(bExecute := FALSE);
END_IF
END_METHOD

END_FUNCTION_BLOCK

// ---- SOURCE/Utilities/Path/FB_PathUtilities.TcPOU
FUNCTION_BLOCK FB_PathUtilities IMPLEMENTS I_Path
VAR_INPUT
END_VAR
VAR_OUTPUT
END_VAR
VAR
	_pathGenerator	: FB_PathGenerator;
END_VAR

(* Checks if path exists, return TRUE when done and the result is returned in `result` output var.*)
METHOD Exists : BOOL
VAR_INPUT
	path	: Tc2_System.T_MaxString;
	netId	: Tc2_System.T_AmsNetID;
END_VAR

VAR_OUTPUT
	result		: BOOL; // Result, if the file exists or not - check when method returns TRUE
	error		: BOOL;	// Will be true if an error occurs while executing the file query
	errorInfo	: ZigaLibs_Core.ST_AdsError; // Error information will be provided here
END_VAR

VAR
	splitPath			: Tc2_System.T_MaxString;
	lastPathPart		: Tc2_System.T_MaxString;
	pathSeperatorLeft	: STRING := '\';
	pathSeperatorRight	: STRING := '/';
	charPosiiton		: INT;
	currentFileEntry	: Tc2_Utilities.ST_FindFileEntry;
	currentSplitString	: Tc2_System.T_MaxString;
	index				: DINT;
END_VAR

VAR_INST
	files				: ARRAY[0..100] OF Tc2_Utilities.ST_FindFileEntry;
	directoryUtilities	 : FB_DirectoryUtilities;
END_VAR
IF directoryUtilities.ListAll(path := path, netId := netId, items :=files, error => error, errorInfo => errorInfo) THEN
	lastPathPart := path;
	
	IF Tc2_Standard.FIND(STR1 := lastPathPart, STR2 := pathSeperatorLeft) <> 0 THEN
		WHILE Tc2_Standard.FIND(STR1 := lastPathPart, STR2 := pathSeperatorLeft) <> 0 DO
			charPosiiton := Tc2_Standard.FIND(lastPathPart, pathSeperatorLeft);
			lastPathPart := Tc2_Standard.DELETE(lastPathPart, charPosiiton, 1);
		END_WHILE		
	ELSIF Tc2_Standard.FIND(STR1 := lastPathPart, STR2 := pathSeperatorRight) <> 0 THEN	
		WHILE Tc2_Standard.FIND(STR1 := lastPathPart, STR2 := pathSeperatorRight) <> 0 DO
			charPosiiton := Tc2_Standard.FIND(lastPathPart, pathSeperatorRight);
			lastPathPart := Tc2_Standard.DELETE(lastPathPart, charPosiiton, 1);
		END_WHILE	
	END_IF
	
	FOR index := 0 TO 100 BY 1 DO
		currentFileEntry := files[index];
		IF currentFileEntry.sFileName = lastPathPart THEN
			result := TRUE;
			EXIT;
		END_IF
	END_FOR

	Exists := TRUE;
END_IF
END_METHOD

(* Generates the file path based on the location, file name and extension*)
METHOD Generate : I_PathGenerator
Generate := _pathGenerator;
END_METHOD

END_FUNCTION_BLOCK

// ---- TESTS/Test suites/FB_Utilities_Tests.TcPOU
FUNCTION_BLOCK INTERNAL FB_Utilities_Tests EXTENDS FB_TestSuite

Test01_ValidateReferences();

METHOD Test01_ValidateReferences
VAR_INPUT
END_VAR
TcUnit.TEST('Test01_ValidateReferences');

AssertTrue(Utilities.Directory <> 0, 'Directory property is not valid!');
AssertTrue(Utilities.File <> 0, 'File property is not valid!');
AssertTrue(Utilities.Path <> 0, 'Path property is not valid!');

TcUnit.TEST_FINISHED();
END_METHOD

END_FUNCTION_BLOCK

// ---- TESTS/Test suites/FB_FileHandler_Tests.TcPOU
// Subject under test
FUNCTION_BLOCK INTERNAL FB_FileHandler_Tests EXTENDS FB_TestSuite

// Create instance variables that will be accesible for all tests
VAR
	_fileHandler								: FB_FileHandler;
	_binaryWriteText							: STRING(300) := 'In a world full of possibilities, every moment is a chance to embrace growth, explore new horizons, and ignite your inner potential. Believe in the power of change, stay curious, and never stop learning. Your journey is unique, and every step forward brings you closer to your dreams.';
	WRITE_TEST_CONTENT_OVERWRITE_EMPTY_FILE 	: Tc2_System.T_MaxString := 'Some random text...';
	WRITE_TEST_CONTENT_APPEND					: Tc2_System.T_MaxString := 'Some more text....';
	WRITE_TEST_CONTENT_OVERWRITE_EXTISTING		: Tc2_System.T_MaxString := 'Only this text should exist...';
	EXPECTED_RESULT_APPEND						: Tc2_System.T_MaxString := 
		Tc2_Standard.CONCAT(WRITE_TEST_CONTENT_OVERWRITE_EMPTY_FILE, WRITE_TEST_CONTENT_APPEND);
END_VAR

VAR CONSTANT
	NEW_TEXT_FILE_NAME		: Tc2_System.T_MaxString := 'FileName.txt';
	NEW_BINARY_FILE_NAME	: Tc2_System.T_MaxString := 'BinaryFileName.txt';
	EXISTING_FILE_NAME		: Tc2_System.T_MaxString := 'ExistingFile.txt';
END_VAR

Test00_Open_NonExistentFile_ExpectError();
Test01_Open_ExistingFile_ExpectNoError_ValidateFileProperty();
Test02_Close_ExpectFileHandleIsZero();
Test03_Create_ExpectFileExists();
Test04_WriteLine_FileNotOpened_ExpectError();
Test05_WriteLine_FileOpened_Overwrite_ExpectNoError_ValidateContent();
Test06_WriteLine_FileOpened_Append_ExpectNoError_ExpectOldAndNewContent();
Test07_WriteLine_FileOpened_Overwrite_ExpectNoError_ExpectOnlyNewContent();
Test08_WriteBinary_FileOpened_Overwrite_ExpectNoError_ExpectOnlyNewContent();
// Append binary does not work - this is a TwinCAT issue...
//Test09_WriteBinary_FileOpened_Append_ExpectNoError_ExpectOldAndNewContent();
Test10_WriteBinary_FileOpened_Overwrite_ExpectNoError_ExpectOnlyNewContent();
Test11_CreateFile_WriteContent_Flush_ExpectFileContent();
Test12_OpenFile_CloseFile_OpenLast_ExpectFileOpened();
CleanupDirectory();

METHOD CleanupDirectory
IF TcUnit.TEST_ORDERED('CleanupDirectory') AND InitTestFolder()  THEN
	IF _fileHandler.File.IsOpened THEN
		_fileHandler.Close();
	ELSIF Utilities.Directory.DeleteFilesCreatedBefore(PRG_TESTS.FILE_HANDLER_TESTS_PATH, '.txt', PRG_TESTS.NET_ID, PRG_TESTS.DATE_TIME_MAX_VALUE) THEN
		TcUnit.TEST_FINISHED();
	END_IF
END_IF
END_METHOD

// Init tests folder with existing file
METHOD PRIVATE InitTestFolder : BOOL
VAR_INST
	initDone	: BOOL;
END_VAR
InitTestFolder := initDone;

IF initDone THEN 
	RETURN;
END_IF

IF _fileHandler.Create(
	path := PRG_TESTS.FILE_HANDLER_TESTS_PATH,
	name := EXISTING_FILE_NAME,
	netId := PRG_TESTS.NET_ID) 
THEN
	initDone := TRUE;
END_IF
END_METHOD

METHOD Test00_Open_NonExistentFile_ExpectError
IF TcUnit.TEST_ORDERED('Test00_Open_NonExistentFile_ExpectError') AND InitTestFolder() THEN
	IF _fileHandler.Open(
		PRG_TESTS.FILE_HANDLER_TESTS_PATH, 
		'I_dont_exist', 
		E_FileOpenMode.BINARY_READ_MUST_EXIST, PRG_TESTS.NET_ID) 
	THEN
		AssertTrue(_fileHandler.Error, 'Opening non existing file should trigger an error');
		AssertEquals_DINT(0, _fileHandler.File.Handle, 'Handle property should be 0.');
		AssertFalse(_fileHandler.File.IsOpened, 'IsOpened property should be FALSE.');
		TcUnit.TEST_FINISHED();
	END_IF
END_IF
END_METHOD

METHOD Test01_Open_ExistingFile_ExpectNoError_ValidateFileProperty
VAR_INPUT
END_VAR
IF TcUnit.TEST_ORDERED('Test01_Open_ExistingFile_ExpectNoError_ValidateFileProperty') AND InitTestFolder()  THEN
	IF _fileHandler.Open(
		PRG_TESTS.FILE_HANDLER_TESTS_PATH, 
		EXISTING_FILE_NAME, 
		E_FileOpenMode.BINARY_READ_MUST_EXIST, PRG_TESTS.NET_ID) 
	THEN
		AssertEquals_STRING(PRG_TESTS.FILE_HANDLER_TESTS_PATH,_fileHandler.File.Path, 'Path property is incorrect');
		AssertEquals_STRING(EXISTING_FILE_NAME,_fileHandler.File.Name, 'Name property is incorrect');
		AssertEquals_STRING(PRG_TESTS.NET_ID,_fileHandler.File.NetId, 'NetId property is incorrect');
		AssertTrue(_fileHandler.File.Handle <> 0, 'Handle property should not be 0.');
		AssertTrue(_fileHandler.File.IsOpened, 'IsOpened property should be TRUE.');
		TcUnit.TEST_FINISHED();
	END_IF
END_IF
END_METHOD

METHOD Test02_Close_ExpectFileHandleIsZero
VAR_INPUT
END_VAR
IF TcUnit.TEST_ORDERED('Test02_Close_ExpectFileHandleIsZero') AND InitTestFolder()  THEN
	IF _fileHandler.Close() THEN
		AssertEquals_uint(0,_fileHandler.File.Handle, 
			'When file is closed, the handle should be 0.');
			
		AssertFalse(_fileHandler.File.IsOpened, 
			'When file is closed, "File.IsOpened" should be FALSE');
			
		_fileHandler.Reset();
		TcUnit.TEST_FINISHED();
	END_IF
END_IF
END_METHOD

METHOD Test03_Create_ExpectFileExists
VAR_INPUT
END_VAR
VAR
	fileExists	: BOOL;
END_VAR
IF TcUnit.TEST_ORDERED('Test03_Create_ExpectFileExists') AND InitTestFolder()  THEN
	IF _fileHandler.Create(PRG_TESTS.FILE_HANDLER_TESTS_PATH, NEW_TEXT_FILE_NAME, PRG_TESTS.NET_ID) THEN
		AssertFalse(_fileHandler.Error, Tc2_Standard.CONCAT('An error occured: ', _fileHandler.AdsError.Message));
		IF Utilities.File.Exists(PRG_TESTS.FILE_HANDLER_TESTS_PATH, NEW_TEXT_FILE_NAME, PRG_TESTS.NET_ID, result => fileExists) THEN
			AssertTrue(fileExists, 'File creation failed, not found.');
			TcUnit.TEST_FINISHED();
		END_IF
	END_IF
END_IF
END_METHOD

METHOD Test04_WriteLine_FileNotOpened_ExpectError
VAR_INPUT
END_VAR
IF TcUnit.TEST_ORDERED('Test04_WriteLine_FileNotOpened_ExpectError') AND InitTestFolder()  THEN
	IF _fileHandler.WriteLine('lallala') THEN
		AssertTrue(_fileHandler.Error, 'Writing to a file if it has not been opened should trigger an error.');
		AssertFalse(_fileHandler.File.IsOpened, 'If file is not opened, the IsOpened should be false!');
		_fileHandler.Reset();
		TcUnit.TEST_FINISHED();
	END_IF
END_IF
END_METHOD

METHOD Test05_WriteLine_FileOpened_Overwrite_ExpectNoError_ValidateContent
VAR_INST
	content		: Tc2_System.T_MaxString;
	state		: INT;
END_VAR
IF TcUnit.TEST_ORDERED('Test05_WriteLine_FileOpened_Overwrite_ExpectNoError_ValidateContent') AND InitTestFolder()  THEN
	CASE state OF
		0:
			IF _fileHandler.Open(PRG_TESTS.FILE_HANDLER_TESTS_PATH, NEW_TEXT_FILE_NAME, E_FileOpenMode.TEXT_READ_WRITE_OVERWRITE_EXISTING, PRG_TESTS.NET_ID) THEN
				state := state + 1;
			END_IF
			
		1:
			IF  _fileHandler.WriteLine(WRITE_TEST_CONTENT_OVERWRITE_EMPTY_FILE)  THEN
				AssertFalse(_filehandler.Error, 'Error writing content...');
				state := state + 1;
			END_IF
		
		2: 
			IF _fileHandler.Close()  THEN
				state := state + 1;
			END_IF
			
		3:
			IF _fileHandler.Open(PRG_TESTS.FILE_HANDLER_TESTS_PATH, NEW_TEXT_FILE_NAME, E_FileOpenMode.TEXT_READ_MUST_EXIST, PRG_TESTS.NET_ID) THEN
				state := state + 1;
			END_IF
			
		4:
			IF _fileHandler.Read(content) THEN
				AssertFalse(_filehandler.Error, 'Error reading content...');
				AssertEquals_STRING(WRITE_TEST_CONTENT_OVERWRITE_EMPTY_FILE, content, 
						'Written content differs.');
				state := state + 1;
			END_IF
			
		5:
			IF _fileHandler.Close() THEN
				TcUnit.TEST_FINISHED();
			END_IF
	END_CASE
END_IF
END_METHOD

METHOD Test06_WriteLine_FileOpened_Append_ExpectNoError_ExpectOldAndNewContent
VAR_INST
	content		: Tc2_System.T_MaxString;
	state		: INT;
END_VAR
IF TcUnit.TEST_ORDERED('Test06_WriteLine_FileOpened_Append_ExpectNoError_ExpectOldAndNewContent') AND InitTestFolder()  THEN
	CASE state OF
		0:
			IF _fileHandler.Open(PRG_TESTS.FILE_HANDLER_TESTS_PATH, NEW_TEXT_FILE_NAME, E_FileOpenMode.TEXT_READ_WRITE_APPEND, PRG_TESTS.NET_ID) THEN
				state := state + 1;
			END_IF
			
		1:
			IF  _fileHandler.WriteLine(WRITE_TEST_CONTENT_APPEND)  THEN
				AssertFalse(_filehandler.Error, 
					Tc2_Standard.CONCAT('Error writing content: ',_fileHandler.AdsError.Message));
				state := state + 1;
			END_IF
		
		2: 
			// Flush the content so that it appears in the file to be read with .Read()
			IF _fileHandler.Flush()  THEN
				state := state + 1;
			END_IF
			
		3:
			IF _fileHandler.Read(content) THEN
				AssertFalse(_filehandler.Error, 
					Tc2_Standard.CONCAT('Error writing content: ',_fileHandler.AdsError.Message));
				AssertEquals_STRING(EXPECTED_RESULT_APPEND, content, 
						'Written content differs.');
				state := state + 1;
			END_IF
			
		4:
			IF _fileHandler.Close() THEN
				TcUnit.TEST_FINISHED();
			END_IF
	END_CASE
END_IF
END_METHOD

METHOD Test07_WriteLine_FileOpened_Overwrite_ExpectNoError_ExpectOnlyNewContent
VAR_INST
	content		: Tc2_System.T_MaxString;
	state		: INT;
END_VAR
IF TcUnit.TEST_ORDERED('Test07_WriteLine_FileOpened_Overwrite_ExpectNoError_ExpectOnlyNewContent') AND InitTestFolder()  THEN
	CASE state OF
		0:
			IF _fileHandler.Open(PRG_TESTS.FILE_HANDLER_TESTS_PATH, NEW_TEXT_FILE_NAME, E_FileOpenMode.TEXT_READ_WRITE_OVERWRITE_EXISTING, PRG_TESTS.NET_ID) THEN
				state := state + 1;
			END_IF
			
		1:
			IF  _fileHandler.WriteLine(WRITE_TEST_CONTENT_OVERWRITE_EXTISTING)  THEN
				AssertFalse(_filehandler.Error, 'Error writing content...');
				state := state + 1;
			END_IF
		
		2: 
			IF _fileHandler.Close()  THEN
				state := state + 1;
			END_IF
			
		3:
			IF _fileHandler.Open(PRG_TESTS.FILE_HANDLER_TESTS_PATH, NEW_TEXT_FILE_NAME, E_FileOpenMode.TEXT_READ_MUST_EXIST, PRG_TESTS.NET_ID) THEN
				state := state + 1;
			END_IF	
			
		4:
			IF _fileHandler.Read(content) THEN
				AssertFalse(_filehandler.Error, 'Error reading content...');
				AssertEquals_STRING(WRITE_TEST_CONTENT_OVERWRITE_EXTISTING, content, 
						'Written content differs.');
				state := state + 1;
			END_IF
			
		5:
			IF _fileHandler.Close() THEN
				TcUnit.TEST_FINISHED();
			END_IF
	END_CASE
END_IF
END_METHOD

METHOD Test08_WriteBinary_FileOpened_Overwrite_ExpectNoError_ExpectOnlyNewContent
VAR_INST
	content		: Tc2_System.T_MaxString;
	state		: INT;
END_VAR
IF TcUnit.TEST_ORDERED('Test08_WriteBinary_FileOpened_Overwrite_ExpectNoError_ExpectOnlyNewContent') AND InitTestFolder()  THEN
	CASE state OF
		0:
			IF _fileHandler.Open(PRG_TESTS.FILE_HANDLER_TESTS_PATH, NEW_BINARY_FILE_NAME, E_FileOpenMode.BINARY_READ_WRITE_OVERWRITE_EXISTING, PRG_TESTS.NET_ID) THEN
				state := state + 1;
			END_IF
			
		1:
			IF _fileHandler.WriteBinary(THIS^.WRITE_TEST_CONTENT_OVERWRITE_EMPTY_FILE)  THEN
				AssertFalse(_filehandler.Error, 'Error writing content...');
				state := state + 1;
			END_IF
		
		2: 
			IF _fileHandler.Close()  THEN
				state := state + 1;
			END_IF
			
		// Open in non-owerwrite mode, otherwise the content is clearly deleted...
		3: 
			IF _fileHandler.Open(PRG_TESTS.FILE_HANDLER_TESTS_PATH, NEW_BINARY_FILE_NAME, E_FileOpenMode.BINARY_READ_WRITE_MUST_EXIST, PRG_TESTS.NET_ID) THEN
				state := state + 1;
			END_IF
			
		4:
			IF _fileHandler.Read(content) THEN
				AssertFalse(_filehandler.Error, 'Error reading content...');
				AssertEquals_STRING(WRITE_TEST_CONTENT_OVERWRITE_EMPTY_FILE, content, 
						'Written content differs.');
				state := state + 1;
			END_IF
			
		5:
			IF _fileHandler.Close() THEN
				TcUnit.TEST_FINISHED();
			END_IF
	END_CASE
END_IF
END_METHOD

METHOD Test09_WriteBinary_FileOpened_Append_ExpectNoError_ExpectOldAndNewContent : REFERENCE TO FB_Test
VAR_INST
	content		: Tc2_System.T_MaxString;
	state		: INT;
END_VAR
IF TcUnit.TEST_ORDERED('Test09_WriteBinary_FileOpened_Append_ExpectNoError_ExpectOldAndNewContent') AND InitTestFolder()  THEN
	CASE state OF
		0:
			IF _fileHandler.Open(PRG_TESTS.FILE_HANDLER_TESTS_PATH, NEW_BINARY_FILE_NAME, E_FileOpenMode.BINARY_APPEND, PRG_TESTS.NET_ID) THEN
				state := state + 1;
			END_IF
			
		1:
			IF  _fileHandler.WriteBinary(WRITE_TEST_CONTENT_APPEND)  THEN
				AssertFalse(_filehandler.Error, 'Error writing content...');
				state := state + 1;
			END_IF
		
		2: 
			IF _fileHandler.Close()  THEN
				state := state + 1;
			END_IF
		
		// Open in non-owerwrite mode, otherwise the content is clearly deleted...
		3: 
			IF _fileHandler.Open(PRG_TESTS.FILE_HANDLER_TESTS_PATH, NEW_BINARY_FILE_NAME, E_FileOpenMode.BINARY_READ_WRITE_MUST_EXIST, PRG_TESTS.NET_ID) THEN
				state := state + 1;
			END_IF

		4:
			IF _fileHandler.Read(content) THEN
				AssertFalse(_filehandler.Error, 'Error reading content...');
				AssertEquals_STRING(EXPECTED_RESULT_APPEND, content, 
						'Written content differs.');
				state := state + 1;
			END_IF
			
		5:
			IF _fileHandler.Close() THEN
				TcUnit.TEST_FINISHED();
			END_IF
	END_CASE
END_IF
END_METHOD

METHOD Test10_WriteBinary_FileOpened_Overwrite_ExpectNoError_ExpectOnlyNewContent : REFERENCE TO FB_Test
VAR_INST
	content		: Tc2_System.T_MaxString;
	state		: INT;
END_VAR
IF TcUnit.TEST_ORDERED('Test10_WriteBinary_FileOpened_Overwrite_ExpectNoError_ExpectOnlyNewContent') AND InitTestFolder()  THEN
CASE state OF
		0:
			IF _fileHandler.Open(PRG_TESTS.FILE_HANDLER_TESTS_PATH, NEW_BINARY_FILE_NAME, E_FileOpenMode.BINARY_READ_WRITE_OVERWRITE_EXISTING, PRG_TESTS.NET_ID) THEN
				state := state + 1;
			END_IF
			
		1:
			IF  _fileHandler.WriteBinary(data := _binaryWriteText)  THEN
				AssertFalse(_filehandler.Error, 'Error writing content...');
				state := state + 1;
			END_IF
		
		2: 
			IF _fileHandler.Close()  THEN
				state := state + 1;
			END_IF
			
		// Open in non-owerwrite mode, otherwise the content is clearly deleted...
		3: 
			IF _fileHandler.Open(PRG_TESTS.FILE_HANDLER_TESTS_PATH, NEW_BINARY_FILE_NAME, E_FileOpenMode.BINARY_READ_WRITE_MUST_EXIST, PRG_TESTS.NET_ID) THEN
				state := state + 1;
			END_IF
			
		4:
			IF _fileHandler.Read(content) THEN
				AssertFalse(_filehandler.Error, 'Error reading content...');
				AssertEquals_STRING(_binaryWriteText, content, 
						'Written content differs.');
				state := state + 1;
			END_IF
			
		5:
			IF _fileHandler.Close() THEN
				TcUnit.TEST_FINISHED();
			END_IF
	END_CASE
END_IF
END_METHOD

METHOD Test11_CreateFile_WriteContent_Flush_ExpectFileContent
VAR_INPUT
END_VAR
VAR_INST
	state	: INT;
	content	: Tc2_System.T_MaxString;
END_VAR
IF TcUnit.TEST_ORDERED('Test11_CreateFile_WriteContent_Flush_ExpectFileContent') AND InitTestFolder()  THEN
	
	CASE state OF
		0:
			IF _fileHandler.Create(PRG_TESTS.FILE_HANDLER_TESTS_PATH, 'FlushTestFile.txt', PRG_TESTS.NET_ID) THEN
				state := state + 1;
			END_IF
			
			
		1:
			IF _fileHandler.Open(PRG_TESTS.FILE_HANDLER_TESTS_PATH, 'FlushTestFile.txt', E_FileOpenMode.TEXT_READ_WRITE_APPEND, PRG_TESTS.NET_ID) THEN
				state := state + 1;
			END_IF
			
		2:
			IF _fileHandler.WriteLine('Some random content....') THEN
				state := state + 1;
			END_IF
			
		3:
			IF _fileHandler.Flush() THEN
				state := state + 1;
			END_IF
			
		4:
			IF _fileHandler.Read(content) THEN
				AssertEquals_STRING('Some random content....', content, 'Content differs');
				AssertFalse(content = '', 'Flushing did not make the file content appear.');
				state := state + 1;
			END_IF
			
		5:
			IF NOT _fileHandler.File.IsOpened OR_ELSE _fileHandler.Close() THEN
				IF Utilities.File.Delete(PRG_TESTS.FILE_HANDLER_TESTS_PATH, 'FlushTestFile.txt', PRG_TESTS.NET_ID) THEN
					TcUnit.TEST_FINISHED();
				END_IF
			END_IF
	END_CASE
END_IF
END_METHOD

METHOD Test12_OpenFile_CloseFile_OpenLast_ExpectFileOpened
VAR_INPUT
END_VAR
VAR_INST
	state	: INT;
END_VAR
IF TcUnit.TEST_ORDERED('Test12_OpenFile_CloseFile_OpenLast_ExpectFileOpened') AND InitTestFolder()  THEN
	CASE state OF
		0: 
			IF _fileHandler.Open(PRG_TESTS.FILE_HANDLER_TESTS_PATH, 'RopenFileTest.txt', E_FileOpenMode.TEXT_READ_WRITE_APPEND, PRG_TESTS.NET_ID) THEN
				state := state + 1;
			END_IF
		
		1:
			IF _fileHandler.Close() THEN
				state := state + 1;
			END_IF
		2:
			IF _fileHandler.OpenLast() THEN
				AssertFalse(_fileHandler.Error, 'Error while opening last file.');
				AssertTrue(_fileHandler.File.IsOpened, 'File should be opened');
				AssertTrue(_fileHandler.File.Handle <> 0, 'File handle should not be 0.');
				state := state + 1;
			END_IF
		
		3:
			IF _fileHandler.Close() THEN
				state := state + 1;
			END_IF
			
		4:
			IF Utilities.File.Delete(_fileHandler.File.Path, _fileHandler.File.Name, PRG_TESTS.NET_ID) THEN
				TcUnit.TEST_FINISHED();
			END_IF
		END_CASE
END_IF
END_METHOD

END_FUNCTION_BLOCK

// ---- TESTS/Test suites/FB_PathUtilities_Tests.TcPOU
FUNCTION_BLOCK INTERNAL FB_PathUtilities_Tests EXTENDS FB_TestSuite
VAR_INPUT
END_VAR
VAR_OUTPUT
END_VAR
VAR
	_pathUtilities	: FB_PathUtilities;
END_VAR

Test01_PathExists();
Test02_PathDoesNotExist_ExpectFalseResult();

METHOD Test01_PathExists
VAR_INPUT
END_VAR
VAR
	exists	: BOOL;
END_VAR
IF TcUnit.TEST_ORDERED('Test01_PathExists') THEN
	IF _pathUtilities.Exists(PRG_TESTS.FILE_HANDLER_TESTS_PATH, PRG_TESTS.NET_ID, result => exists) THEN
		AssertTrue(exists, 'Provided path exists, returned result should be TRUE');
		TcUnit.TEST_FINISHED();
	END_IF
END_IF
END_METHOD

METHOD Test02_PathDoesNotExist_ExpectFalseResult
VAR_INPUT
END_VAR
VAR
	exists	: BOOL;
END_VAR
IF TcUnit.TEST_ORDERED('Test02_PathDoesNotExist_ExpectFalseResult') THEN
	IF _pathUtilities.Exists('Some randome path...', '', result => exists) THEN
		AssertFalse(exists, 'Provided path does not exist, returned result should be FALSE.');
		TcUnit.TEST_FINISHED();
	END_IF
END_IF
END_METHOD

END_FUNCTION_BLOCK

// ---- TESTS/Test suites/FB_FileUtilities_Tests.TcPOU
FUNCTION_BLOCK INTERNAL FB_FileUtilities_Tests EXTENDS TcUnit.FB_TestSuite
VAR_INPUT
END_VAR
VAR_OUTPUT
END_VAR
VAR
	_fileUtilities	: FB_FileUtilities;
END_VAR
VAR CONSTANT
	FILE_NAME	: Tc2_System.T_MaxString := 'FileUtilitiesCreateTestFile.txt';
END_VAR

Test01_CreateFile_ExpectNoError();
Test02_Exists_ValidateCreatedFileExists();
Test03_DeleteFile_ExpectFileNoLongerExists();

METHOD Test01_CreateFile_ExpectNoError
VAR_INPUT
END_VAR
VAR
	error		: BOOL;
	errorInfo	: ZigaLibs_Core.ST_AdsError;
END_VAR
IF TcUnit.TEST_ORDERED('Test01_CreateFile_ExpectNoError') THEN
	IF _fileUtilities.Create(PRG_TESTS.FILE_HANDLER_TESTS_PATH, FILE_NAME, PRG_TESTS.NET_ID, FALSE, error => error, errorInfo => errorInfo) OR error THEN
		AssertFalse(error, Tc2_Standard.CONCAT('Unexpected error occured while creating file.', errorInfo.Message));
		TcUnit.TEST_FINISHED();
	END_IF
END_IF
END_METHOD

METHOD Test02_Exists_ValidateCreatedFileExists
VAR_INPUT
END_VAR

VAR
	exists		: BOOL;
	error		: BOOL;
	errorInfo	: ZigaLibs_Core.ST_AdsError;
END_VAR
IF TcUnit.TEST_ORDERED('Test02_Exists_ValidateCreatedFileExists') THEN
	IF _fileUtilities.Exists(PRG_TESTS.FILE_HANDLER_TESTS_PATH, FILE_NAME, '', result => exists,error => error, errorInfo => errorInfo) THEN
		AssertTrue(exists, 'Created file should exist.');
		AssertFalse(error, Tc2_Standard.CONCAT('Unexpected error occurred while checking file existion: ', errorInfo.Message));
		TcUnit.TEST_FINISHED();
	END_IF
END_IF
END_METHOD

METHOD Test03_DeleteFile_ExpectFileNoLongerExists
VAR_INPUT
END_VAR
VAR_INST
	error			: BOOL;
	errorInfo		: ZigaLibs_Core.ST_AdsError;
	fileDeleteDone	: BOOL;
	fileExists		: BOOL;
END_VAR
IF TcUnit.TEST_ORDERED('Test03_DeleteFile_ExpectFileNoLongerExists') THEN
	IF NOT fileDeleteDone AND_THEN 
		_fileUtilities.Delete(PRG_TESTS.FILE_HANDLER_TESTS_PATH, FILE_NAME, PRG_TESTS.NET_ID, error => error, errorInfo => errorInfo) 
	THEN
		AssertFalse(error, Tc2_Standard.CONCAT('Unexpected error occurred while deleting file: ', errorInfo.Message));
		fileDeleteDone := TRUE;
	ELSIF fileDeleteDone THEN
		IF _fileUtilities.Exists(PRG_TESTS.FILE_HANDLER_TESTS_PATH, FILE_NAME, PRG_TESTS.NET_ID, result => fileExists) THEN
			AssertFalse(fileExists, 'File still exists, deletion failed.');
			TcUnit.TEST_FINISHED();
		END_IF
	END_IF
END_IF
END_METHOD

END_FUNCTION_BLOCK

// ---- TESTS/Test suites/FB_DirectoryUtilities_Tests.TcPOU
FUNCTION_BLOCK INTERNAL FB_DirectoryUtilities_Tests EXTENDS FB_TestSuite
VAR_INPUT
END_VAR
VAR_OUTPUT
END_VAR
VAR
	_directoryUtilities	: FB_DirectoryUtilities;
END_VAR

Test01_CreateFile_Wait3Seconds_DeleteWithFileCreatedBeforeMethod();
Test02_TryDeletingButNoFilesMatchCriteria_ExpectNoErrors();

METHOD Test01_CreateFile_Wait3Seconds_DeleteWithFileCreatedBeforeMethod
VAR_INPUT
END_VAR
VAR_INST
	fileCreated			: BOOL;
	delayForDelete		: Tc2_Standard.TON;
	currentSystemTime	: DT;
	getSystemTime		: Tc2_System.GETSYSTEMTIME;
	fileTime			: Tc2_Utilities.T_FILETIME;
	dateTime			: DT;
	dtUpperLimit  		: DT  := DATE_AND_TIME#2106-02-07-06:28:15;
	error				: BOOL;
	errorInfo			: ZigaLibs_Core.ST_AdsError;
	deletedFiles		: ARRAY[0..100] OF Tc2_System.T_MaxString;
END_VAR
IF TcUnit.TEST_ORDERED('Test01_CreateFile_Wait3Seconds_DeleteWithFileCreatedBeforeMethod') THEN
	IF NOT fileCreated THEN
		IF Utilities.File.Create(PRG_TESTS.FILE_HANDLER_TESTS_PATH, 'FileToDeleteViaDeleteBeforeMethod.txt', '', FALSE, 
			error => error ,errorInfo => errorInfo)
		THEN
			fileCreated := TRUE;
			AssertFalse(error, Tc2_Standard.CONCAT('Unexpected error when creating the file: ', errorInfo.Message));
		END_IF
	ELSE
		delayForDelete(IN := TRUE, PT := T#3S);
		IF delayForDelete.Q THEN
			getSystemTime(timeHiDW => fileTime.dwHighDateTime, timeLoDW => fileTime.dwLowDateTime);
			IF _directoryUtilities.DeleteFilesCreatedBefore(PRG_TESTS.FILE_HANDLER_TESTS_PATH, 'FileToDeleteViaDeleteBeforeMet', '', dtUpperLimit, 
				error=> error, errorInfo => errorInfo, deletedFiles => deletedFiles)
			THEN
				AssertTrue(deletedFiles[0] = 'FileToDeleteViaDeleteBeforeMethod.txt', 'Deleted files list contains no items!');
				AssertFalse(error, Tc2_Standard.CONCAT('Deleting files encountered an undexpected error: ', errorInfo.Message));
				TcUnit.TEST_FINISHED();
			END_IF
		END_IF
	END_IF
END_IF
END_METHOD

METHOD Test02_TryDeletingButNoFilesMatchCriteria_ExpectNoErrors
VAR_INPUT
END_VAR
VAR_INST
	fileTime			: Tc2_Utilities.T_FILETIME;
	dateTime			: DT;
	dtUpperLimit  		: DT  := DATE_AND_TIME#2106-02-07-06:28:15;
	error				: BOOL;
	errorInfo			: ZigaLibs_Core.ST_AdsError;
	deletedFiles		: ARRAY[0..100] OF Tc2_System.T_MaxString;
END_VAR
IF TcUnit.TEST_ORDERED('Test02_TryDeletingButNoFilesMatchCriteria_ExpectNoErrors') THEN
	IF Utilities.Directory.DeleteFilesCreatedBefore(PRG_TESTS.FILE_HANDLER_TESTS_PATH, 'MyLog', PRG_TESTS.NET_ID, dtUpperLimit, 
				error=> error, errorInfo => errorInfo, deletedFiles => deletedFiles) THEN
	AssertFalse(error, 'An error has happened attempting to call the DeleteFilesCreatedBefore with no matching content provided.');
	TcUnit.TEST_FINISHED();
	END_IF
END_IF
END_METHOD

END_FUNCTION_BLOCK
